REGION Network 74: Good Count 3
   RUNG wire#powerrail
      Contact( "Unit1.Em6.ControlNodes".cmHotPressLeftServoPress.monitoring.resultOK )
      Contact( "Unit1.Em6.ControlNodes".cmHotPressLeftServoPress.monitoring.complete )
      wire#w1
      P_Trig( #citi_Ptrig[3] )
      Coil( "Unit1.Em6.ControlNodes".citiMap.PMC.Machining_Assembly.IncrGood_Count )
   END_RUNG
   RUNG wire#powerrail
      Contact( #citiTest[3] )
   END_RUNG wire#w1
   // the same network as SCL:
   #_w1 := ("Unit1.Em6.ControlNodes".cmHotPressLeftServoPress.monitoring.resultOK AND "Unit1.Em6.ControlNodes".cmHotPressLeftServoPress.monitoring.complete) OR #citiTest[3];
   #_w2 := #_w1 AND NOT #citi_Ptrig[3];   // rising edge
   #citi_Ptrig[3] := #_w1;
   "Unit1.Em6.ControlNodes".citiMap.PMC.Machining_Assembly.IncrGood_Count := #_w2;
END_REGION

REGION Network 75: Reject Count 4 X
   RUNG wire#powerrail
      Contact( "Unit1.Em6.ControlNodes".cmHotPressLeftServoPress.monitoring.resultNG )
      Contact( "Unit1.Em6.ControlNodes".cmHotPressLeftServoPress.monitoring.complete )
      wire#w1
      P_Trig( #citi_Ptrig[4] )
      Coil( "Unit1.Em6.ControlNodes".citiMap.PMC.Machining_Assembly.IncrReject_Count )
   END_RUNG
   RUNG wire#powerrail
      Contact( #citiTest[4] )
   END_RUNG wire#w1
   // the same network as SCL:
   #_w1 := ("Unit1.Em6.ControlNodes".cmHotPressLeftServoPress.monitoring.resultNG AND "Unit1.Em6.ControlNodes".cmHotPressLeftServoPress.monitoring.complete) OR #citiTest[4];
   #_w2 := #_w1 AND NOT #citi_Ptrig[4];   // rising edge
   #citi_Ptrig[4] := #_w1;
   "Unit1.Em6.ControlNodes".citiMap.PMC.Machining_Assembly.IncrReject_Count := #_w2;
END_REGION

REGION Network 76: Cycle End Trigger 5
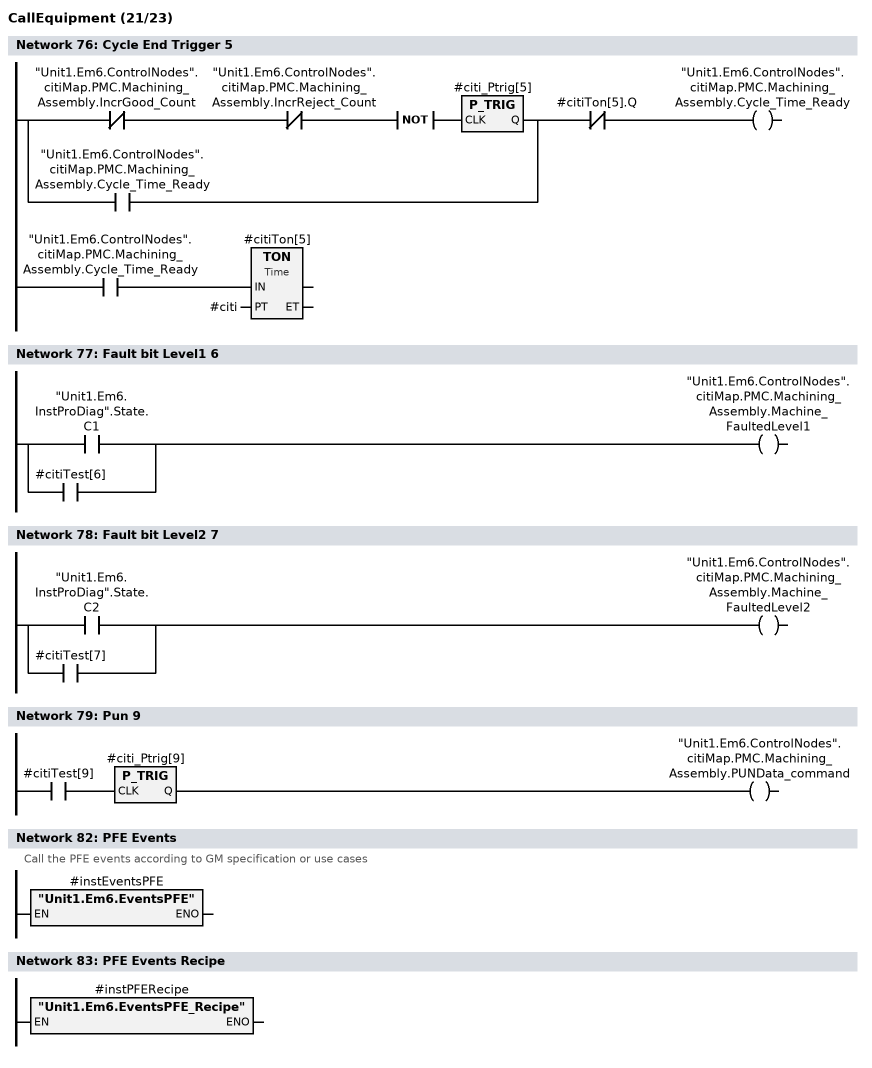
   RUNG wire#powerrail
      I_Contact( "Unit1.Em6.ControlNodes".citiMap.PMC.Machining_Assembly.IncrGood_Count )
      I_Contact( "Unit1.Em6.ControlNodes".citiMap.PMC.Machining_Assembly.IncrReject_Count )
      Not()
      P_Trig( #citi_Ptrig[5] )
      wire#w1
      I_Contact( #citiTon[5].Q )
      Coil( "Unit1.Em6.ControlNodes".citiMap.PMC.Machining_Assembly.Cycle_Time_Ready )
   END_RUNG
   RUNG wire#powerrail
      Contact( "Unit1.Em6.ControlNodes".citiMap.PMC.Machining_Assembly.Cycle_Time_Ready )
   END_RUNG wire#w1
   RUNG wire#powerrail
      Contact( "Unit1.Em6.ControlNodes".citiMap.PMC.Machining_Assembly.Cycle_Time_Ready )
      { S7_Templates := "time_type := Time" } #citiTon[5].TON(pt := #citi, et =>)
   END_RUNG
   // the same network as SCL:
   #_w1 := NOT (NOT "Unit1.Em6.ControlNodes".citiMap.PMC.Machining_Assembly.IncrGood_Count AND NOT "Unit1.Em6.ControlNodes".citiMap.PMC.Machining_Assembly.IncrReject_Count);
   #_w2 := #_w1 AND NOT #citi_Ptrig[5];   // rising edge
   #citi_Ptrig[5] := #_w1;
   "Unit1.Em6.ControlNodes".citiMap.PMC.Machining_Assembly.Cycle_Time_Ready := (#_w2 OR "Unit1.Em6.ControlNodes".citiMap.PMC.Machining_Assembly.Cycle_Time_Ready) AND NOT #citiTon[5].Q;
   #citiTon[5].TON(IN := "Unit1.Em6.ControlNodes".citiMap.PMC.Machining_Assembly.Cycle_Time_Ready, PT := #citi);
END_REGION

REGION Network 77: Fault bit Level1 6
   RUNG wire#powerrail
      Contact( "Unit1.Em6.InstProDiag".State.C1 )
      wire#w1
      Coil( "Unit1.Em6.ControlNodes".citiMap.PMC.Machining_Assembly.Machine_FaultedLevel1 )
   END_RUNG
   RUNG wire#powerrail
      Contact( #citiTest[6] )
   END_RUNG wire#w1
   // the same network as SCL:
   "Unit1.Em6.ControlNodes".citiMap.PMC.Machining_Assembly.Machine_FaultedLevel1 := "Unit1.Em6.InstProDiag".State.C1 OR #citiTest[6];
END_REGION

REGION Network 78: Fault bit Level2 7
   RUNG wire#powerrail
      Contact( "Unit1.Em6.InstProDiag".State.C2 )
      wire#w1
      Coil( "Unit1.Em6.ControlNodes".citiMap.PMC.Machining_Assembly.Machine_FaultedLevel2 )
   END_RUNG
   RUNG wire#powerrail
      Contact( #citiTest[7] )
   END_RUNG wire#w1
   // the same network as SCL:
   "Unit1.Em6.ControlNodes".citiMap.PMC.Machining_Assembly.Machine_FaultedLevel2 := "Unit1.Em6.InstProDiag".State.C2 OR #citiTest[7];
END_REGION

REGION Network 79: Pun 9
   RUNG wire#powerrail
      Contact( #citiTest[9] )
      P_Trig( #citi_Ptrig[9] )
      Coil( "Unit1.Em6.ControlNodes".citiMap.PMC.Machining_Assembly.PUNData_command )
   END_RUNG
   // the same network as SCL:
   #_w1 := #citiTest[9] AND NOT #citi_Ptrig[9];   // rising edge
   #citi_Ptrig[9] := #citiTest[9];
   "Unit1.Em6.ControlNodes".citiMap.PMC.Machining_Assembly.PUNData_command := #_w1;
END_REGION

REGION Network 81: ******************** PFE Events ********************
END_REGION

REGION Network 82: PFE Events
   // Call the PFE events according to GM specification or use cases
   RUNG wire#powerrail
      #instEventsPFE()
   END_RUNG
   // the same network as SCL:
   #instEventsPFE();   // "Unit1.Em6.EventsPFE"
END_REGION

REGION Network 83: PFE Events Recipe
   RUNG wire#powerrail
      #instPFERecipe()
   END_RUNG
   // the same network as SCL:
   #instPFERecipe();   // "Unit1.Em6.EventsPFE_Recipe"
END_REGION

REGION Network 84: ************************ Part Result Data ************************
END_REGION

REGION Network 85: Hot Press Left Results Data
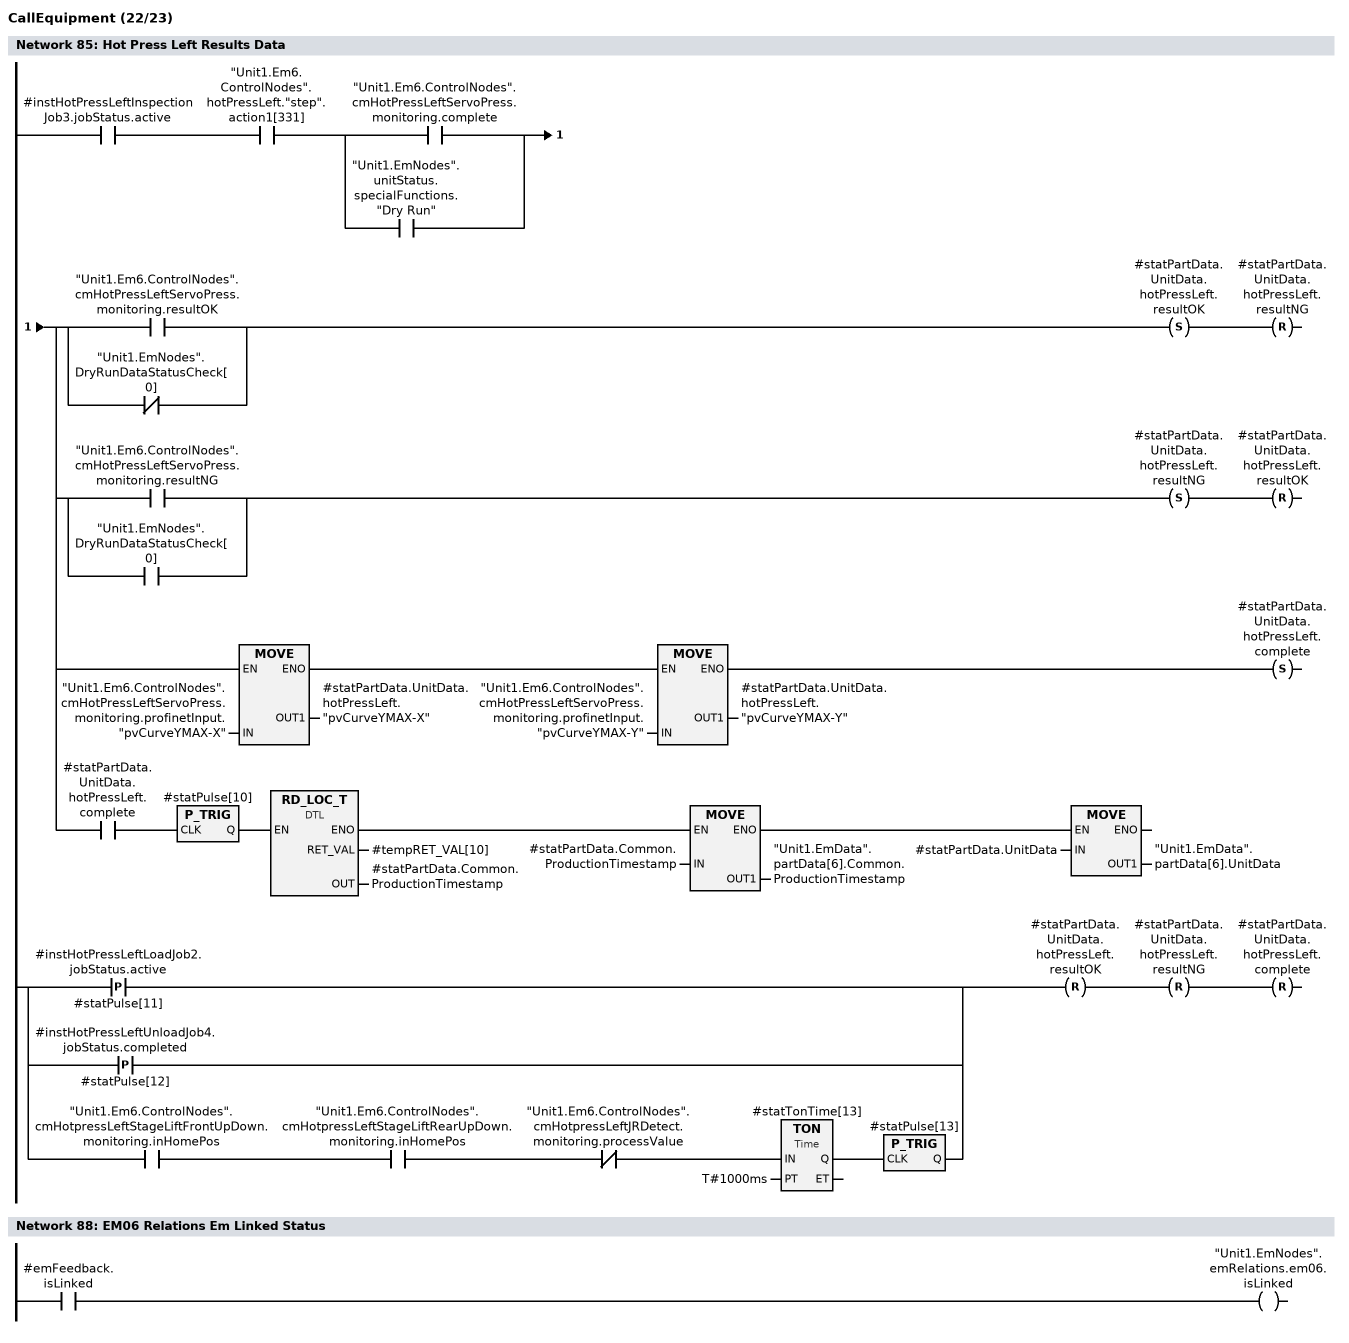
   RUNG wire#powerrail
      Contact( #instHotPressLeftInspectionJob3.jobStatus.active )
      Contact( "Unit1.Em6.ControlNodes".hotPressLeft."step".action1[331] )
      wire#w1
      Contact( "Unit1.Em6.ControlNodes".cmHotPressLeftServoPress.monitoring.complete )
      wire#w2
      Contact( "Unit1.Em6.ControlNodes".cmHotPressLeftServoPress.monitoring.resultOK )
      wire#w3
      S_Coil( #statPartData.UnitData.hotPressLeft.resultOK )
      R_Coil( #statPartData.UnitData.hotPressLeft.resultNG )
   END_RUNG
   RUNG wire#w1
      Contact( "Unit1.EmNodes".unitStatus.specialFunctions."Dry Run" )
   END_RUNG wire#w2
   RUNG wire#w2
      I_Contact( "Unit1.EmNodes".DryRunDataStatusCheck[0] )
   END_RUNG wire#w3
   RUNG wire#w2
      Contact( "Unit1.Em6.ControlNodes".cmHotPressLeftServoPress.monitoring.resultNG )
      wire#w4
      S_Coil( #statPartData.UnitData.hotPressLeft.resultNG )
      R_Coil( #statPartData.UnitData.hotPressLeft.resultOK )
   END_RUNG
   RUNG wire#w2
      Contact( "Unit1.EmNodes".DryRunDataStatusCheck[0] )
   END_RUNG wire#w4
   RUNG wire#w2
      Move(in := "Unit1.Em6.ControlNodes".cmHotPressLeftServoPress.monitoring.profinetInput."pvCurveYMAX-X", out1 => #statPartData.UnitData.hotPressLeft."pvCurveYMAX-X")
      Move(in := "Unit1.Em6.ControlNodes".cmHotPressLeftServoPress.monitoring.profinetInput."pvCurveYMAX-Y", out1 => #statPartData.UnitData.hotPressLeft."pvCurveYMAX-Y")
      S_Coil( #statPartData.UnitData.hotPressLeft.complete )
   END_RUNG
   RUNG wire#w2
      Contact( #statPartData.UnitData.hotPressLeft.complete )
      P_Trig( #statPulse[10] )
      { S7_Templates := "date_type := DTL" } RD_LOC_T(RET_VAL => #tempRET_VAL[10], OUT => #statPartData.Common.ProductionTimestamp)
      Move(in := #statPartData.Common.ProductionTimestamp, out1 => "Unit1.EmData".partData[6].Common.ProductionTimestamp)
      Move(in := #statPartData.UnitData, out1 => "Unit1.EmData".partData[6].UnitData)
   END_RUNG
   RUNG wire#powerrail
      P_Contact(operand := #instHotPressLeftLoadJob2.jobStatus.active, bit := #statPulse[11])
      wire#w5
      R_Coil( #statPartData.UnitData.hotPressLeft.resultOK )
      R_Coil( #statPartData.UnitData.hotPressLeft.resultNG )
      R_Coil( #statPartData.UnitData.hotPressLeft.complete )
   END_RUNG
   RUNG wire#powerrail
      P_Contact(operand := #instHotPressLeftUnloadJob4.jobStatus.completed, bit := #statPulse[12])
   END_RUNG wire#w5
   RUNG wire#powerrail
      Contact( "Unit1.Em6.ControlNodes".cmHotpressLeftStageLiftFrontUpDown.monitoring.inHomePos )
      Contact( "Unit1.Em6.ControlNodes".cmHotpressLeftStageLiftRearUpDown.monitoring.inHomePos )
      I_Contact( "Unit1.Em6.ControlNodes".cmHotpressLeftJRDetect.monitoring.processValue )
      { S7_Templates := "time_type := Time" } #statTonTime[13].TON(pt := T#1000ms, et =>)
      P_Trig( #statPulse[13] )
   END_RUNG wire#w5
   // the same network as SCL:
   #_w1 := #instHotPressLeftInspectionJob3.jobStatus.active AND "Unit1.Em6.ControlNodes".hotPressLeft."step".action1[331] AND ("Unit1.Em6.ControlNodes".cmHotPressLeftServoPress.monitoring.complete OR "Unit1.EmNodes".unitStatus.specialFunctions."Dry Run");
   IF #_w1 AND ("Unit1.Em6.ControlNodes".cmHotPressLeftServoPress.monitoring.resultOK OR NOT "Unit1.EmNodes".DryRunDataStatusCheck[0]) THEN
       #statPartData.UnitData.hotPressLeft.resultOK := TRUE;
       #statPartData.UnitData.hotPressLeft.resultNG := FALSE;
   END_IF;
   IF #_w1 AND ("Unit1.Em6.ControlNodes".cmHotPressLeftServoPress.monitoring.resultNG OR "Unit1.EmNodes".DryRunDataStatusCheck[0]) THEN
       #statPartData.UnitData.hotPressLeft.resultNG := TRUE;
       #statPartData.UnitData.hotPressLeft.resultOK := FALSE;
   END_IF;
   IF #_w1 THEN
       #statPartData.UnitData.hotPressLeft."pvCurveYMAX-X" := "Unit1.Em6.ControlNodes".cmHotPressLeftServoPress.monitoring.profinetInput."pvCurveYMAX-X";
       #statPartData.UnitData.hotPressLeft."pvCurveYMAX-Y" := "Unit1.Em6.ControlNodes".cmHotPressLeftServoPress.monitoring.profinetInput."pvCurveYMAX-Y";
       #statPartData.UnitData.hotPressLeft.complete := TRUE;
   END_IF;
   #_w2 := #_w1 AND #statPartData.UnitData.hotPressLeft.complete;
   #_w3 := #_w2 AND NOT #statPulse[10];   // rising edge
   #statPulse[10] := #_w2;
   #tempRET_VAL[10] := RD_LOC_T(EN := #_w3, OUT => #statPartData.Common.ProductionTimestamp, ENO => #_w4);
   IF #_w4 THEN
       "Unit1.EmData".partData[6].Common.ProductionTimestamp := #statPartData.Common.ProductionTimestamp;
       "Unit1.EmData".partData[6].UnitData := #statPartData.UnitData;
   END_IF;
   #_w5 := #instHotPressLeftLoadJob2.jobStatus.active AND NOT #statPulse[11];   // rising edge of #instHotPressLeftLoadJob2.jobStatus.active
   #statPulse[11] := #instHotPressLeftLoadJob2.jobStatus.active;
   #_w6 := #instHotPressLeftUnloadJob4.jobStatus.completed AND NOT #statPulse[12];   // rising edge of #instHotPressLeftUnloadJob4.jobStatus.completed
   #statPulse[12] := #instHotPressLeftUnloadJob4.jobStatus.completed;
   #statTonTime[13].TON(IN := "Unit1.Em6.ControlNodes".cmHotpressLeftStageLiftFrontUpDown.monitoring.inHomePos AND "Unit1.Em6.ControlNodes".cmHotpressLeftStageLiftRearUpDown.monitoring.inHomePos AND NOT "Unit1.Em6.ControlNodes".cmHotpressLeftJRDetect.monitoring.processValue,
                        PT := T#1000ms);
   #_w7 := #statTonTime[13].Q AND NOT #statPulse[13];   // rising edge
   #statPulse[13] := #statTonTime[13].Q;
   IF #_w5 OR #_w6 OR #_w7 THEN
       #statPartData.UnitData.hotPressLeft.resultOK := FALSE;
       #statPartData.UnitData.hotPressLeft.resultNG := FALSE;
       #statPartData.UnitData.hotPressLeft.complete := FALSE;
   END_IF;
END_REGION

REGION Network 87: ************************ Unit Output ************************
END_REGION

REGION Network 88: EM06 Relations Em Linked Status
   RUNG wire#powerrail
      Contact( #emFeedback.isLinked )
      Coil( "Unit1.EmNodes".emRelations.em06.isLinked )
   END_RUNG
   // the same network as SCL:
   "Unit1.EmNodes".emRelations.em06.isLinked := #emFeedback.isLinked;
END_REGION

REGION Network 89: Em6 Relations Em State
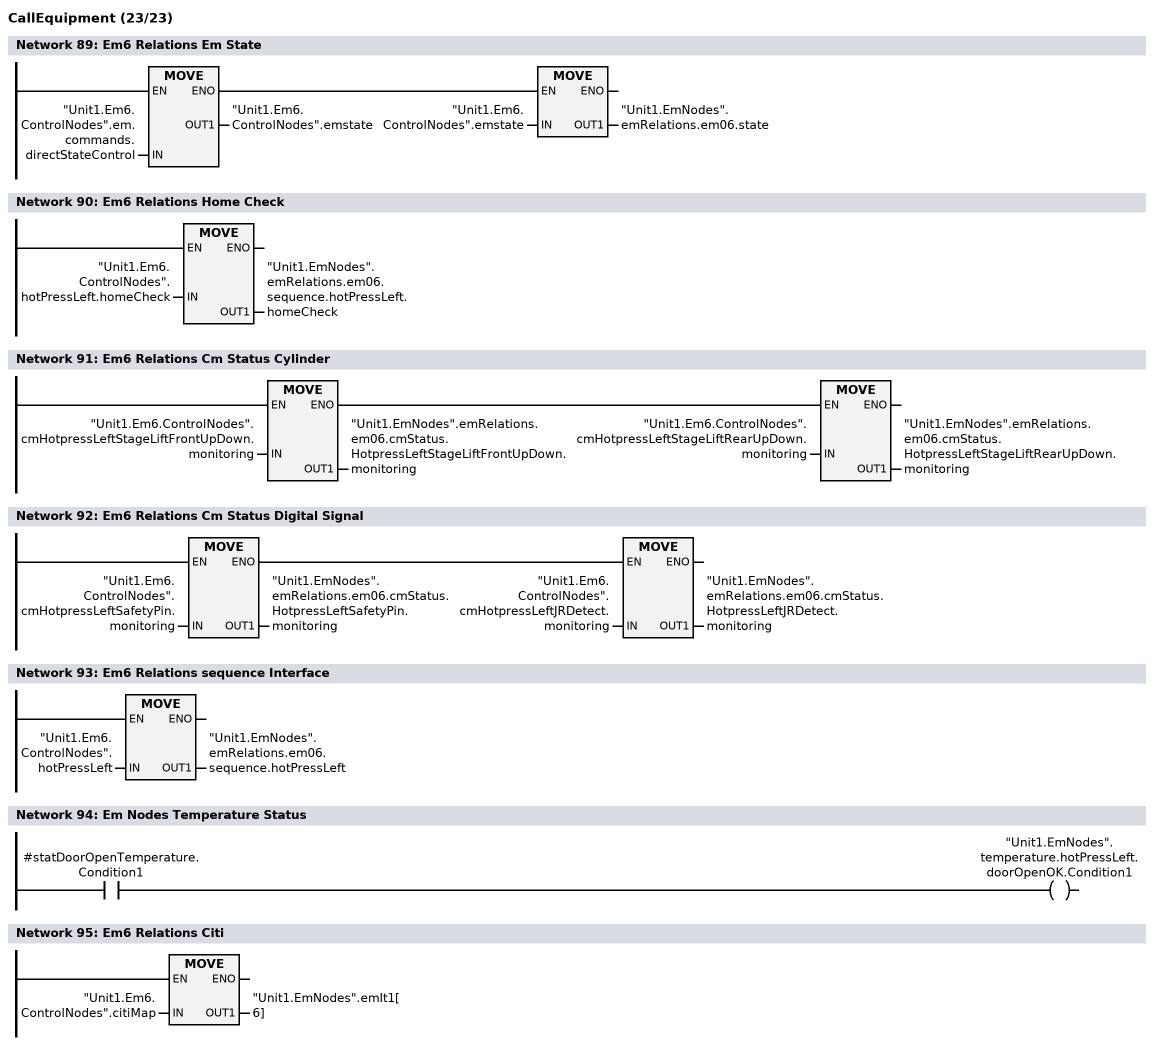
   RUNG wire#powerrail
      Move(in := "Unit1.Em6.ControlNodes".em.commands.directStateControl, out1 => "Unit1.Em6.ControlNodes".emstate)
      Move(in := "Unit1.Em6.ControlNodes".emstate, out1 => "Unit1.EmNodes".emRelations.em06.state)
   END_RUNG
   // the same network as SCL:
   "Unit1.Em6.ControlNodes".emstate := "Unit1.Em6.ControlNodes".em.commands.directStateControl;
   "Unit1.EmNodes".emRelations.em06.state := "Unit1.Em6.ControlNodes".emstate;
END_REGION

REGION Network 90: Em6 Relations Home Check
   RUNG wire#powerrail
      Move(in := "Unit1.Em6.ControlNodes".hotPressLeft.homeCheck, out1 => "Unit1.EmNodes".emRelations.em06.sequence.hotPressLeft.homeCheck)
   END_RUNG
   // the same network as SCL:
   "Unit1.EmNodes".emRelations.em06.sequence.hotPressLeft.homeCheck := "Unit1.Em6.ControlNodes".hotPressLeft.homeCheck;
END_REGION

REGION Network 91: Em6 Relations Cm Status Cylinder
   RUNG wire#powerrail
      Move(in := "Unit1.Em6.ControlNodes".cmHotpressLeftStageLiftFrontUpDown.monitoring, out1 => "Unit1.EmNodes".emRelations.em06.cmStatus.HotpressLeftStageLiftFrontUpDown.monitoring)
      Move(in := "Unit1.Em6.ControlNodes".cmHotpressLeftStageLiftRearUpDown.monitoring, out1 => "Unit1.EmNodes".emRelations.em06.cmStatus.HotpressLeftStageLiftRearUpDown.monitoring)
   END_RUNG
   // the same network as SCL:
   "Unit1.EmNodes".emRelations.em06.cmStatus.HotpressLeftStageLiftFrontUpDown.monitoring := "Unit1.Em6.ControlNodes".cmHotpressLeftStageLiftFrontUpDown.monitoring;
   "Unit1.EmNodes".emRelations.em06.cmStatus.HotpressLeftStageLiftRearUpDown.monitoring := "Unit1.Em6.ControlNodes".cmHotpressLeftStageLiftRearUpDown.monitoring;
END_REGION

REGION Network 92: Em6 Relations Cm Status Digital Signal
   RUNG wire#powerrail
      Move(in := "Unit1.Em6.ControlNodes".cmHotpressLeftSafetyPin.monitoring, out1 => "Unit1.EmNodes".emRelations.em06.cmStatus.HotpressLeftSafetyPin.monitoring)
      Move(in := "Unit1.Em6.ControlNodes".cmHotpressLeftJRDetect.monitoring, out1 => "Unit1.EmNodes".emRelations.em06.cmStatus.HotpressLeftJRDetect.monitoring)
   END_RUNG
   // the same network as SCL:
   "Unit1.EmNodes".emRelations.em06.cmStatus.HotpressLeftSafetyPin.monitoring := "Unit1.Em6.ControlNodes".cmHotpressLeftSafetyPin.monitoring;
   "Unit1.EmNodes".emRelations.em06.cmStatus.HotpressLeftJRDetect.monitoring := "Unit1.Em6.ControlNodes".cmHotpressLeftJRDetect.monitoring;
END_REGION

REGION Network 93: Em6 Relations sequence Interface
   RUNG wire#powerrail
      Move(in := "Unit1.Em6.ControlNodes".hotPressLeft, out1 => "Unit1.EmNodes".emRelations.em06.sequence.hotPressLeft)
   END_RUNG
   // the same network as SCL:
   "Unit1.EmNodes".emRelations.em06.sequence.hotPressLeft := "Unit1.Em6.ControlNodes".hotPressLeft;
END_REGION

REGION Network 94: Em Nodes Temperature Status
   RUNG wire#powerrail
      Contact( #statDoorOpenTemperature.Condition1 )
      Coil( "Unit1.EmNodes".temperature.hotPressLeft.doorOpenOK.Condition1 )
   END_RUNG
   // the same network as SCL:
   "Unit1.EmNodes".temperature.hotPressLeft.doorOpenOK.Condition1 := #statDoorOpenTemperature.Condition1;
END_REGION

REGION Network 95: Em6 Relations Citi
   RUNG wire#powerrail
      Move(in := "Unit1.Em6.ControlNodes".citiMap, out1 => "Unit1.EmNodes".emIt1[6])
   END_RUNG
   // the same network as SCL:
   "Unit1.EmNodes".emIt1[6] := "Unit1.Em6.ControlNodes".citiMap;
END_REGION
END_FUNCTION_BLOCK
